FUNCTION_BLOCK InjectorController
  (* Standard: 61499-2 *)
  (* Version 0.1, 2016-00-28, hpea485, UOA *)
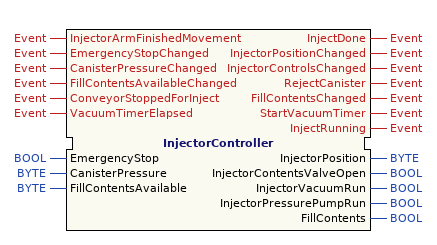
  EVENT_INPUT
    InjectorArmFinishedMovement;
    EmergencyStopChanged;
    CanisterPressureChanged;
    FillContentsAvailableChanged;
    ConveyorStoppedForInject;
    VacuumTimerElapsed;
  END_EVENT
  EVENT_OUTPUT
    InjectDone;
    InjectorPositionChanged;
    InjectorControlsChanged;
    RejectCanister;
    FillContentsChanged;
    StartVacuumTimer;
    InjectRunning;
  END_EVENT
  VAR_INPUT
    EmergencyStop : BOOL;
    CanisterPressure : BYTE;
    FillContentsAvailable : BYTE;
  END_VAR
  VAR_OUTPUT
    InjectorPosition : BYTE;
    InjectorContentsValveOpen : BOOL;
    InjectorVacuumRun : BOOL;
    InjectorPressurePumpRun : BOOL;
    FillContents : BOOL;
  END_VAR
  FBS
    Arm : InjectorMotorController;
    Pumps : InjectorPumpsController;
  END_FBS
  EVENT_CONNECTIONS
    InjectorArmFinishedMovement TO Arm.InjectorArmFinishedMovement;
    EmergencyStopChanged TO Arm.EmergencyStopChanged;
    EmergencyStopChanged TO Pumps.EmergencyStopChanged;
    CanisterPressureChanged TO Pumps.CanisterPressureChanged;
    FillContentsAvailableChanged TO Pumps.FillContentsAvailableChanged;
    ConveyorStoppedForInject TO Arm.ConveyorStoppedForInject;
    VacuumTimerElapsed TO Pumps.VacuumTimerElapsed;
    Arm.InjectDone TO InjectDone;
    Arm.InjectorPositionChanged TO InjectorPositionChanged;
    Pumps.InjectorControlsChanged TO InjectorControlsChanged;
    Pumps.RejectCanister TO RejectCanister;
    Pumps.FillContentsChanged TO FillContentsChanged;
    Pumps.StartVacuumTimer TO StartVacuumTimer;
    Arm.InjectRunning TO InjectRunning;
    Arm.StartPump TO Pumps.StartPump;
    Pumps.PumpFinished TO Arm.PumpFinished;
  END_CONNECTIONS
  DATA_CONNECTIONS
    EmergencyStop TO Arm.EmergencyStop;
    EmergencyStop TO Pumps.EmergencyStop;
    CanisterPressure TO Pumps.CanisterPressure;
    FillContentsAvailable TO Pumps.FillContentsAvailable;
    Arm.InjectorPosition TO InjectorPosition;
    Pumps.InjectorContentsValveOpen TO InjectorContentsValveOpen;
    Pumps.InjectorVacuumRun TO InjectorVacuumRun;
    Pumps.InjectorPressurePumpRun TO InjectorPressurePumpRun;
    Pumps.FillContents TO FillContents;
  END_CONNECTIONS
END_FUNCTION_BLOCK
